PROGRAM PRG_Test
VAR
	fbSensorTest			: FB_SensorTest;
	fbElectrovalveTest		: FB_ElectroValveTest;
	fbButtontest			: FB_ButtonTest;
	fbLapmBlinkingTest		: FB_LampBlinkingTest;
	
	fbActuatortest			: FB_ActuatorTest;
	
	fbSensortestDecoratorTest	: FB_Sensor_DecoratorTestTest;
	
	fbActuator_TestDecoratorWithoutTimeTest	: FB_Actuator_TestDecoratorWithoutTimeTest;
	fbActuator_TestDecoratorWithTimeTest	: FB_Actuator_TestDecoratorWithTimeTest;
	
END_VAR


	TcUnit.RUN_IN_SEQUENCE ();


GVL_Variable.fbSaveDataByADS (
	bWrite		:= GVL_Variable.bSave,
	sNetId		:= ,
	nPort		:= ,
	sVarName	:= GVL_Variable.sData,
	nSrcAddr	:= ADR (GVL_Variable.bValueToSave),
	nLen		:= SIZEOF (GVL_Variable.bValueToSave),
	tTimeout	:= ,
	eComMode	:= ,
	bBusy		=> GVL_Variable.bSaved,
	bError		=> ,
	nErrorId	=>
);

END_PROGRAM

(* stored: Version 1.1.0.1
   POU PRG_Test: Id {1d1ad101-c2d4-0277-1bb3-7445680eebd7}, SpecialFunc None *)
